FUNCTION_BLOCK SHARED_COMPRESSOR (* Extracted Composite Function Block Type *)
  (* Standard: 61499-2 *)
  (* Version 4/29/2023, Dmitrii *)
  PACKAGE UAO.Hackathon;
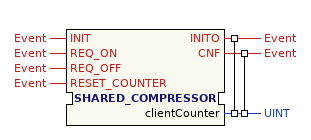
  EVENT_INPUT
    INIT; (* Init *)
    REQ_ON; (* Increment 'on' counter *)
    REQ_OFF; (* Decrement 'on' counter *)
    RESET_COUNTER; (* Reset counter *)
  END_EVENT
  EVENT_OUTPUT
    INITO WITH clientCounter; (* Initialization confirm *)
    CNF WITH clientCounter; (* Execution Confirmation *)
  END_EVENT
  VAR_OUTPUT
    clientCounter : UINT;
  END_VAR
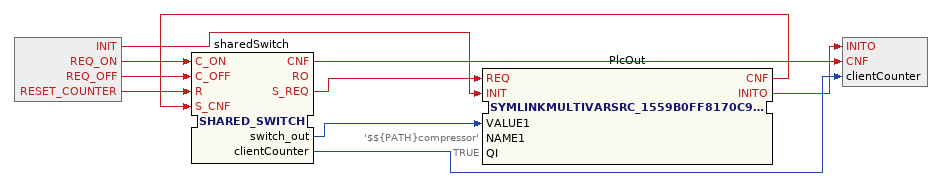
  FBS
    PlcOut : SYMLINKMULTIVARSRC_1559B0FF8170C9BA0(NAME1 := '$${PATH}compressor', QI := TRUE); {SET_ATTRIBUTE(Configuration.GenericFBType.InterfaceParams, Runtime.System#I:=1;VALUE${I$}:BOOL)}
    sharedSwitch : SHARED_SWITCH;
  END_FBS
  EVENT_CONNECTIONS
    sharedSwitch.S_REQ TO PlcOut.REQ;
    PlcOut.CNF TO sharedSwitch.S_CNF;
    PlcOut.INITO TO INITO;
    REQ_ON TO sharedSwitch.C_ON;
    REQ_OFF TO sharedSwitch.C_OFF;
    RESET_COUNTER TO sharedSwitch.R;
    INIT TO PlcOut.INIT;
    sharedSwitch.CNF TO CNF;
  END_CONNECTIONS
  DATA_CONNECTIONS
    sharedSwitch.switch_out TO PlcOut.VALUE1;
    sharedSwitch.clientCounter TO clientCounter;
  END_CONNECTIONS
END_FUNCTION_BLOCK
